Fanuc KAREL source: ko00093.KL

PROGRAM KO00093
%STACKSIZE=65535
%PRIORITY=65535
%NOLOCKGROUP
VAR
P1 : JOINTPOS9
P2 : JOINTPOS9
F : BOOLEAN
OUT : POSITION
BEGIN
F=TRUE
-- UNSAFE_SOURCE_IR line 11: CALL_RESULT MIRROR(convert_jointpos9_to_xyzwprext(P1), convert_jointpos9_to_position(P2), F)
END KO00093
